Yaskawa INFORM job: OK_R2_O25(90,90)OKKR.JBI

/JOB
//NAME OK_R2_O25(90,90)OKKR
///FOLDERNAME X4
//POS
///NPOS 97,97,97,5,0,0
///TOOL 0
///POSTYPE PULSE
///PULSE
C00000=50835,-53294,-56898,34013,98451,-41646
C00001=66247,-59875,-54045,33572,88031,-38570
C00002=78429,-58697,-57800,22918,88804,-33875
C00003=78429,-58481,-56464,22917,88147,-34001
C00004=78298,-58728,-57763,23043,88768,-33927
C00005=69643,-52105,-49625,33763,92396,-40613
C00006=70861,-53766,-50563,33745,91680,-40337
C00007=69643,-52105,-49625,33763,92396,-40613
C00008=63351,-67995,-58075,33653,87757,-39820
C00009=64656,-67213,-53597,33676,85263,-40042
C00010=65856,-65059,-52521,33643,85160,-39588
C00011=64656,-67213,-53597,33676,85263,-40042
C00012=63351,-67995,-58075,33653,87757,-39820
C00013=45726,-92330,-71384,33030,91093,-45927
C00014=124640,-141323,-85615,30079,47037,-26254
C00015=130744,-1241,-38327,-11105,91766,3467
C00016=129102,16023,-13406,-31158,87839,15094
C00017=123860,36791,4019,-24112,94444,11118
C00018=123804,31839,136,-24116,91545,11670
C00019=123804,31612,1202,-24099,90836,11812
C00020=123804,31839,136,-24116,91545,11670
C00021=123482,33886,2197,-24055,91257,11613
C00022=123804,31839,136,-24116,91545,11670
C00023=125345,30839,-799,-26337,95487,22898
C00024=124720,30743,-895,-26255,95305,22711
C00025=125345,30839,-799,-26337,95487,22898
C00026=129572,22111,-16154,-26217,102424,15263
C00027=134432,-74321,-93176,-21371,80106,4897
C00028=134444,-76872,-84143,-21905,73701,6074
C00029=49509,-92451,-71436,18371,72002,-24485
C00030=70995,-73599,-63483,-5261,57588,4258
C00031=66514,-55217,-53825,-869,65392,2316
C00032=65482,-51746,-52435,104,67666,1944
C00033=65482,-51518,-50928,105,66856,1943
C00034=65482,-51746,-52435,104,67666,1944
C00035=64067,-49440,-51105,623,68038,1432
C00036=67579,-59810,-55128,-3548,59339,2843
C00037=66476,-70430,-60523,-3095,57161,2474
C00038=58197,-65987,-52684,6296,54996,-5238
C00039=59340,-64248,-51807,5712,55263,-4754
C00040=58197,-65987,-52684,6296,54996,-5238
C00041=63788,-69829,-55553,-1849,54329,1451
C00042=56826,-85471,-68230,1656,54084,-1417
C00043=56826,-85471,-68230,1656,54084,-1417
C00044=102451,-13110,-36135,16567,57993,-49425
C00045=109958,-1865,-17297,20837,50330,-58748
C00046=106882,1917,-13595,28180,53287,-63091
C00047=106882,1960,-12459,28418,52686,-63271
C00048=106908,1918,-13088,28273,53002,-63164
C00049=107377,4243,-11107,27998,52825,-62999
C00050=107018,-122,-15473,28061,53338,-63012
C00051=108068,-547,-15827,27421,52993,-62628
C00052=107053,-149,-15797,27976,53491,-62950
C00053=111931,-2152,-16379,18085,49070,-58298
C00054=110631,5617,-7956,11824,43044,-61353
C00055=104636,-10918,-31211,15368,49705,-63104
C00056=108483,-1019,-17560,35302,47868,-72900
C00057=109692,-2140,-18586,34446,47427,-72438
C00058=104713,-2787,-21119,37129,50480,-73783
C00059=102007,-17480,-40404,16896,52392,-63839
C00060=74569,-98048,-84705,40385,49273,-78120
C00061=84906,-149835,-99714,49305,31488,-82745
C00062=67141,-64181,-58377,-15172,73422,22226
C00063=67153,-63147,-54223,-15332,71466,22481
C00064=67158,-63957,-54295,-15365,71109,22532
C00065=68249,-64616,-54976,-15617,71394,22894
C00066=67159,-63511,-55670,-15277,72147,22395
C00067=67988,-62385,-53738,-15523,71717,22756
C00068=70448,-57226,-50975,-16018,73109,23469
C00069=67153,-63147,-54223,-15332,71466,22481
C00070=67141,-63168,-54233,-15330,71460,22478
C00071=39299,-107327,-82845,4045,81700,-26502
C00072=66887,-63669,-54491,21302,99716,-56800
C00073=66885,-63675,-54495,21301,99715,-56801
C00074=67262,-63679,-54113,21334,99394,-56720
C00075=66886,-64055,-55950,21357,100370,-56682
C00076=65816,-62172,-53718,21176,100267,-57098
C00077=68034,-62282,-53641,21471,99592,-56398
C00078=72060,-53392,-48791,22097,99997,-54828
C00079=66885,-63675,-54495,21301,99715,-56801
C00080=45726,-92330,-71384,33030,91093,-45927
C00081=124640,-141323,-85615,30079,47037,-26254
C00082=130744,-1241,-38327,-11105,91766,3467
C00083=129102,16023,-13406,-31158,87839,15094
C00084=124880,28190,-3075,-25525,90475,12377
C00085=123715,29659,118,-25246,89080,12219
C00086=127713,31630,3688,-26474,85269,14457
C00087=129644,30530,3868,-27487,82369,15856
C00088=127309,27205,-10871,-20460,92899,4236
C00089=127809,9858,-27074,-20606,94007,4216
C00090=123663,27737,-5726,-27376,86572,26839
C00091=123538,28089,-4861,-27351,86219,26878
C00092=122504,28004,-4942,-27086,85903,26579
C00093=128085,16419,-15976,-28476,88415,28001
C00094=136273,11855,-27077,-30231,101403,21866
C00095=152636,-99249,-95800,-30488,94254,30020
C00096=51465,-66777,-57067,18771,103495,-61871
BC00000=25181,438263,219567
BC00001=25181,438263,219567
BC00002=25181,438263,219567
BC00003=25181,438263,219567
BC00004=25181,438263,219567
BC00005=25181,438263,219567
BC00006=25181,438263,219567
BC00007=25181,438263,219567
BC00008=25181,438263,219567
BC00009=25181,438263,219567
BC00010=25181,438263,219567
BC00011=25181,438263,219567
BC00012=25181,438263,219567
BC00013=25181,438263,219567
BC00014=2835,438263,219564
BC00015=2835,367555,219564
BC00016=2835,367555,219564
BC00017=2835,367555,219564
BC00018=2835,367555,219564
BC00019=2835,367555,219564
BC00020=2835,367555,219564
BC00021=2835,367555,219564
BC00022=2835,367555,219564
BC00023=2835,367555,219564
BC00024=2835,367555,219564
BC00025=2835,367555,219564
BC00026=2835,367555,219564
BC00027=2835,367555,219564
BC00028=2835,513435,219564
BC00029=133008,437778,302599
BC00030=244352,437277,218186
BC00031=244352,437277,218186
BC00032=244352,437277,218186
BC00033=244352,437277,218186
BC00034=244352,437277,218186
BC00035=244352,437277,218186
BC00036=244352,437277,218186
BC00037=244352,437277,218186
BC00038=244352,437277,218186
BC00039=244352,437277,218186
BC00040=244352,437277,218186
BC00041=244352,437277,218186
BC00042=244352,437277,218186
BC00043=394860,437277,218186
BC00044=394860,389827,218186
BC00045=394860,382020,218186
BC00046=394860,382020,218186
BC00047=394860,382020,218186
BC00048=394860,382020,218186
BC00049=394860,382020,218186
BC00050=394860,382020,218186
BC00051=394860,382020,218186
BC00052=394860,382020,218186
BC00053=394860,382020,218186
BC00054=394860,382020,218186
BC00055=394860,382020,329166
BC00056=394860,382020,329166
BC00057=394860,382020,329166
BC00058=394860,382020,329166
BC00059=394860,382020,218186
BC00060=394860,382020,218186
BC00061=368580,477394,218186
BC00062=238562,403379,275704
BC00063=244169,402720,256754
BC00064=246412,402456,249174
BC00065=246412,402456,249174
BC00066=246412,402456,249174
BC00067=246412,402456,249174
BC00068=246416,397848,249159
BC00069=244179,391506,256717
BC00070=238571,392166,275667
BC00071=135476,398025,275806
BC00072=31317,403944,275946
BC00073=25704,403275,257017
BC00074=23459,403007,249445
BC00075=23459,403007,249445
BC00076=23459,403007,249445
BC00077=23459,403007,249445
BC00078=23459,403007,249445
BC00079=25714,392199,256980
BC00080=25181,438263,219567
BC00081=2835,438263,219564
BC00082=2835,367555,219564
BC00083=2835,367555,219564
BC00084=2835,367555,219564
BC00085=2835,367555,219564
BC00086=2835,367555,219564
BC00087=2835,367555,219564
BC00088=2835,367555,219564
BC00089=2835,367555,344273
BC00090=2835,367555,344273
BC00091=2835,367555,344273
BC00092=2835,367555,344273
BC00093=2835,367555,344273
BC00094=2835,367555,355083
BC00095=2835,493869,355083
BC00096=66280,463284,275909
EC00000=-798156,-740307
EC00001=-798156,-740307
EC00002=-798156,-740307
EC00003=-798156,-740307
EC00004=-798156,-740307
EC00005=-798156,-740307
EC00006=-798156,-740307
EC00007=-798156,-740307
EC00008=-798156,-740307
EC00009=-798156,-740307
EC00010=-798156,-740307
EC00011=-798156,-740307
EC00012=-798156,-740307
EC00013=-798156,-740307
EC00014=-798153,-740307
EC00015=-798153,-740307
EC00016=-798153,-740307
EC00017=-798153,-740307
EC00018=-798153,-740307
EC00019=-798153,-740307
EC00020=-798153,-740307
EC00021=-798153,-740307
EC00022=-798153,-740307
EC00023=-798153,-740307
EC00024=-798153,-740307
EC00025=-798153,-740307
EC00026=-798153,-740307
EC00027=-798153,-740307
EC00028=-798153,-740307
EC00029=-798156,-740307
EC00030=-798156,-740307
EC00031=-798156,-740307
EC00032=-798156,-740307
EC00033=-798156,-740307
EC00034=-798156,-740307
EC00035=-798156,-740307
EC00036=-798156,-740307
EC00037=-798156,-740307
EC00038=-798156,-740307
EC00039=-798156,-740307
EC00040=-798156,-740307
EC00041=-798156,-740307
EC00042=-798156,-740307
EC00043=-798156,-740307
EC00044=-798156,-740307
EC00045=-798156,-740307
EC00046=-798156,-740307
EC00047=-798156,-740307
EC00048=-798156,-740307
EC00049=-798156,-740307
EC00050=-798156,-740307
EC00051=-798156,-740307
EC00052=-798156,-740307
EC00053=-798156,-740307
EC00054=-798156,-740307
EC00055=-798156,-740307
EC00056=-798156,-740307
EC00057=-798156,-740307
EC00058=-798156,-740307
EC00059=-798156,-740307
EC00060=-798156,-740307
EC00061=-798156,-740307
EC00062=-798156,-740307
EC00063=-798156,-740307
EC00064=-798156,-740307
EC00065=-798156,-740307
EC00066=-798156,-740307
EC00067=-798156,-740307
EC00068=-798156,-740307
EC00069=-798156,-740307
EC00070=-798156,-740307
EC00071=-798156,-740307
EC00072=-798156,-740307
EC00073=-798156,-740307
EC00074=-798156,-740307
EC00075=-798156,-740307
EC00076=-798156,-740307
EC00077=-798156,-740307
EC00078=-798156,-740307
EC00079=-798156,-740307
EC00080=-798156,-740307
EC00081=-798153,-740307
EC00082=-798153,-740307
EC00083=-798153,-740307
EC00084=-798153,-740307
EC00085=-798153,-740307
EC00086=-798153,-740307
EC00087=-798153,-740307
EC00088=-798153,-740307
EC00089=-798153,-740307
EC00090=-798153,-740307
EC00091=-798153,-740307
EC00092=-798153,-740307
EC00093=-798153,-740307
EC00094=-798153,-740307
EC00095=-798153,-740307
EC00096=-798156,-740307
///POSTYPE BASE
///RECTAN
///RCONF 0,0,0,0,1,0,0,0,0,0,0,0,0,0,0,0,0,0,0,0,0,0,0,0
P00006=2.006,1.622,-0.565,0.0000,0.0000,0.0000
P00021=0.073,2.058,-0.109,0.0000,0.0000,0.0000
P00022=2.006,1.622,-0.565,0.0000,0.0000,0.0000
///RCONF 0,0,0,0,0,0,0,0,0,0,0,0,0,0,0,0,0,0,0,0,0,0,0,0
P00050=-0.123,2.174,-1.314,0.0000,0.0000,0.0000
P00051=-5.945,4.696,-10.293,0.0000,0.0000,0.0000
//INST
///DATE 2024/11/20 10:49
///ATTR SC,RW
///GROUP1 RB1,BS1
///GROUP2 ST1
NOP
'OK_r2_O25(90,90)
'Path S1039
SFTOF3D
MOVJ C00000 BC00000 VJ=100.00  +MOVJ EC00000 VJ=100.00
MOVL C00001 BC00001 V=400.0  +MOVJ EC00001 VJ=100.00
SMOVL C00002 BC00002 V=100.0  +MOVJ EC00002
SREFP 3 C00003 BC00003  +REFP EC00003
CALL JOB:SEARCH-R1-S13D
SET P022 P006
SFTON3D P022
SMOVL C00004 BC00004 V=100.0  +MOVJ EC00004
SMOVL C00005 BC00005 V=100.0  +MOVJ EC00005
SREFP 3 C00006 BC00006  +REFP EC00006
CALL JOB:SEARCH-R1-S13D
SET P022 P006
SFTON3D P022
SMOVL C00007 BC00007 V=100.0  +MOVJ EC00007
SMOVL C00008 BC00008 V=100.0  +MOVJ EC00008
SMOVL C00009 BC00009 V=100.0  +MOVJ EC00009
SREFP 3 C00010 BC00010  +REFP EC00010
CALL JOB:SEARCH-R1-S13D
SET P022 P006
SFTON3D P022
SMOVL C00011 BC00011 V=100.0  +MOVJ EC00011
SMOVL C00012 BC00012 V=100.0  +MOVJ EC00012
SMOVL C00013 BC00013 V=1000.0  +MOVJ EC00013
MOVJ C00014 BC00014 VJ=100.00  +MOVJ EC00014 VJ=20.00
MOVJ C00015 BC00015 VJ=100.00  +MOVJ EC00015 VJ=20.00
MOVJ C00016 BC00016 VJ=100.00  +MOVJ EC00016 VJ=20.00
SFTOF3D
SMOVL C00017 BC00017 V=250.0  +MOVJ EC00017
SMOVL C00018 BC00018 V=100.0  +MOVJ EC00018
SREFP 3 C00019 BC00019  +REFP EC00019
CALL JOB:SEARCH-R1-S13D
SET P051 P006
SFTON3D P051
SMOVL C00020 BC00020 V=100.0  +MOVJ EC00020
SREFP 3 C00021 BC00021  +REFP EC00021
CALL JOB:SEARCH-R1-S13D
SET P051 P006
SFTON3D P051
SMOVL C00022 BC00022 V=100.0  +MOVJ EC00022
SMOVL C00023 BC00023 V=133.3  +MOVJ EC00023
SREFP 3 C00024 BC00024  +REFP EC00024
CALL JOB:SEARCH-R1-S13D
SET P051 P006
SFTON3D P051
SFTOF3D
SMOVL C00025 BC00025 V=100.0  +MOVJ EC00025
SMOVL C00026 BC00026 V=250.0  +MOVJ EC00026
'DODAC SEARCH
MOVJ C00027 BC00027 VJ=100.00  +MOVJ EC00027 VJ=20.00
MOVJ C00028 BC00028 VJ=100.00  +MOVJ EC00028 VJ=20.00
MOVJ C00029 BC00029 VJ=100.00  +MOVJ EC00029 VJ=100.00
'Path S1430
SFTOF3D
MOVJ C00030 BC00030 VJ=100.00  +MOVJ EC00030 VJ=100.00
MOVL C00031 BC00031 V=166.7  +MOVJ EC00031 VJ=100.00
SMOVL C00032 BC00032 V=100.0  +MOVJ EC00032
SREFP 3 C00033 BC00033  +REFP EC00033
CALL JOB:SEARCH-R1-S13D
SET P021 P006
SFTON3D P021
SMOVL C00034 BC00034 V=100.0  +MOVJ EC00034
SREFP 3 C00035 BC00035  +REFP EC00035
CALL JOB:SEARCH-R1-S13D
SET P021 P006
SFTON3D P021
SMOVL C00036 BC00036 V=100.0  +MOVJ EC00036
SMOVL C00037 BC00037 V=100.0  +MOVJ EC00037
SMOVL C00038 BC00038 V=100.0  +MOVJ EC00038
SREFP 3 C00039 BC00039  +REFP EC00039
CALL JOB:SEARCH-R1-S13D
SET P021 P006
SFTON3D P021
SFTOF3D
SMOVL C00040 BC00040 V=100.0  +MOVJ EC00040
MOVL C00041 BC00041 V=400.0  +MOVJ EC00041 VJ=100.00
MOVL C00042 BC00042 V=1000.0  +MOVJ EC00042 VJ=100.00
MOVJ C00043 BC00043 VJ=100.00  +MOVJ EC00043 VJ=20.00
MOVJ C00044 BC00044 VJ=100.00  +MOVJ EC00044 VJ=20.00
MOVJ C00045 BC00045 VJ=100.00  +MOVJ EC00045 VJ=20.00
SMOVL C00046 BC00046 V=133.3  +MOVJ EC00046
SREFP 3 C00047 BC00047  +REFP EC00047
CALL JOB:SEARCH-R1-S13D
SET P050 P006
SFTON3D P050
SMOVL C00048 BC00048 V=100.0  +MOVJ EC00048
SREFP 3 C00049 BC00049  +REFP EC00049
CALL JOB:SEARCH-R1-S13D
SET P050 P006
SFTON3D P050
SMOVL C00050 BC00050 V=100.0  +MOVJ EC00050
SREFP 3 C00051 BC00051  +REFP EC00051
CALL JOB:SEARCH-R1-S13D
SET P050 P006
SFTON3D P050
SMOVL C00052 BC00052 V=166.7  +MOVJ EC00052
MACRO1 MJ#(0) ARGF14
SMOVL C00053 BC00053 V=166.5  +MOVJ EC00053
ARCON
SMOVL C00054 BC00054 V=7.5  +MOVJ EC00054
ARCOF
MOVJ C00055 BC00055 VJ=100.00  +MOVJ EC00055 VJ=20.00
MACRO1 MJ#(0) ARGF14
SMOVL C00056 BC00056 V=166.7  +MOVJ EC00056
ARCON
SMOVL C00057 BC00057 V=8.3  +MOVJ EC00057
ARCOF
SMOVL C00058 BC00058 V=166.7  +MOVJ EC00058
MOVJ C00059 BC00059 VJ=100.00  +MOVJ EC00059 VJ=20.00
SFTOF3D
MOVJ C00060 BC00060 VJ=100.00  +MOVJ EC00060 VJ=20.00
MOVJ C00061 BC00061 VJ=100.00  +MOVJ EC00061 VJ=20.00
'Path W1431
SFTOF3D
SFTON3D P021
MOVJ C00062 BC00062 VJ=100.00  +MOVJ EC00062 VJ=100.00
SMOVL C00063 BC00063 V=250.0  +MOVJ EC00063
SMOVL C00064 BC00064 V=100.0 PL=0  +MOVJ EC00064
SREFP 1 C00065 BC00065  +REFP EC00065
SREFP 2 C00066 BC00066  +REFP EC00066
MACRO1 MJ#(0) ARGF9
ARCON
SMOVL C00067 BC00067 V=9.2  +MOVJ EC00067
SMOVL C00068 BC00068 V=9.2  +MOVJ EC00068
ARCOF
SMOVL C00069 BC00069 V=400.0  +MOVJ EC00069
SMOVL C00070 BC00070 V=1000.0  +MOVJ EC00070
SFTOF3D
MOVJ C00071 BC00071 VJ=100.00  +MOVJ EC00071 VJ=100.00
'Path W243
SFTOF3D
SFTON3D P022
MOVJ C00072 BC00072 VJ=100.00  +MOVJ EC00072 VJ=100.00
SMOVL C00073 BC00073 V=400.0  +MOVJ EC00073
SMOVL C00074 BC00074 V=133.3 PL=0  +MOVJ EC00074
SREFP 1 C00075 BC00075  +REFP EC00075
SREFP 2 C00076 BC00076  +REFP EC00076
MACRO1 MJ#(0) ARGF9
ARCON
SMOVL C00077 BC00077 V=9.2  +MOVJ EC00077
SMOVL C00078 BC00078 V=9.2  +MOVJ EC00078
ARCOF
SMOVL C00079 BC00079 V=400.0  +MOVJ EC00079
SMOVL C00080 BC00080 V=1000.0  +MOVJ EC00080
MOVJ C00081 BC00081 VJ=100.00  +MOVJ EC00081 VJ=20.00
MOVJ C00082 BC00082 VJ=100.00  +MOVJ EC00082 VJ=20.00
MOVJ C00083 BC00083 VJ=100.00  +MOVJ EC00083 VJ=20.00
SFTOF3D
SMOVL C00084 BC00084 V=250.0  +MOVJ EC00084
MACRO1 MJ#(0) ARGF9
SFTON3D P051
SMOVL C00085 BC00085 V=133.3  +MOVJ EC00085
ARCON
SMOVL C00086 BC00086 V=8.3  +MOVJ EC00086
SMOVL C00087 BC00087 V=8.3  +MOVJ EC00087
ARCOF
SMOVL C00088 BC00088 V=166.7  +MOVJ EC00088
SMOVL C00089 BC00089 V=1000.0  +MOVJ EC00089
SMOVL C00090 BC00090 V=400.0  +MOVJ EC00090
MACRO1 MJ#(0) ARGF14
SMOVL C00091 BC00091 V=166.7  +MOVJ EC00091
ARCON
SMOVL C00092 BC00092 V=8.3  +MOVJ EC00092
ARCOF
SMOVL C00093 BC00093 V=166.7  +MOVJ EC00093
SFTOF3D
MOVJ C00094 BC00094 VJ=100.00  +MOVJ EC00094 VJ=20.00
MOVJ C00095 BC00095 VJ=100.00  +MOVJ EC00095 VJ=20.00
MOVJ C00096 BC00096 VJ=100.00  +MOVJ EC00096 VJ=100.00
SFTOF3D
END
